ABB RAPID module: Codigo Rapid Module1

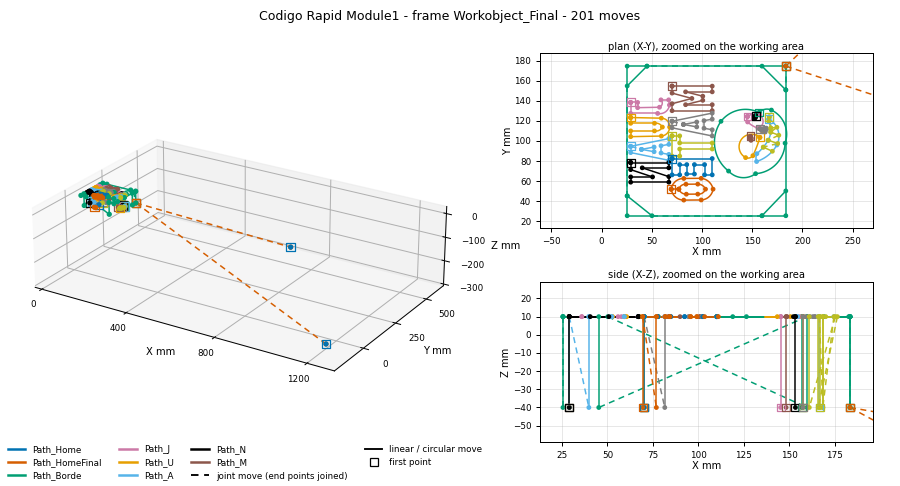
[picture p0: tool path of Codigo Rapid Module1 in frame Workobject_Final, 201 of 201 moves have a stored position in this frame; points joined in program order, loops and branches not executed]
MODULE Module1
    CONST robtarget Target_10:=[[183.5,174.5,-40],[1,0,0,0],[-2,-1,0,0],[9E+09,9E+09,9E+09,9E+09,9E+09,9E+09]];
    CONST robtarget Target_20:=[[183.5,174.5,10],[1,0,0,0],[-2,-1,0,0],[9E+09,9E+09,9E+09,9E+09,9E+09,9E+09]];
    CONST robtarget Target_30:=[[25.5,174.5,10],[1,0,0,0],[-2,-1,0,0],[9E+09,9E+09,9E+09,9E+09,9E+09,9E+09]];
    CONST robtarget Target_40:=[[25.5,25.5,10],[1,0,0,0],[-2,-1,0,0],[9E+09,9E+09,9E+09,9E+09,9E+09,9E+09]];
    CONST robtarget Target_50:=[[183.5,25.5,10],[1,0,0,0],[-2,-1,0,0],[9E+09,9E+09,9E+09,9E+09,9E+09,9E+09]];
    CONST robtarget Target_Home:=[[1257.383388943,-178.562274595,-229.244724109],[0.000082309,-0.261784185,0.00007376,-0.965126431],[0,-1,0,0],[9E+09,9E+09,9E+09,9E+09,9E+09,9E+09]];
    CONST robtarget Target_60:=[[183.5,150.793,-40],[1,0,0,0],[-2,-1,0,0],[9E+09,9E+09,9E+09,9E+09,9E+09,9E+09]];
    CONST robtarget Target_70:=[[183.5,150.793,10],[1,0,0,0],[-2,-1,0,0],[9E+09,9E+09,9E+09,9E+09,9E+09,9E+09]];
    CONST robtarget Target_80:=[[159.793,174.5,10],[1,0,0,0],[-2,-1,0,0],[9E+09,9E+09,9E+09,9E+09,9E+09,9E+09]];
    CONST robtarget Target_90:=[[45.207,174.5,-40],[1,0,0,0],[-2,-1,0,0],[9E+09,9E+09,9E+09,9E+09,9E+09,9E+09]];
    CONST robtarget Target_100:=[[45.207,174.5,10],[1,0,0,0],[-2,-1,0,0],[9E+09,9E+09,9E+09,9E+09,9E+09,9E+09]];
    CONST robtarget Target_110:=[[25.5,154.793,10],[1,0,0,0],[-2,-1,0,0],[9E+09,9E+09,9E+09,9E+09,9E+09,9E+09]];
    CONST robtarget Target_120:=[[25.5,45.24,-40],[1,0,0,0],[-2,-1,0,0],[9E+09,9E+09,9E+09,9E+09,9E+09,9E+09]];
    CONST robtarget Target_130:=[[25.5,45.24,10],[1,0,0,0],[-2,-1,0,0],[9E+09,9E+09,9E+09,9E+09,9E+09,9E+09]];
    CONST robtarget Target_140:=[[50.175,25.5,10],[1,0,0,0],[-2,-1,0,0],[9E+09,9E+09,9E+09,9E+09,9E+09,9E+09]];
    CONST robtarget Target_150:=[[159.787,25.5,-40],[1,0,0,0],[-2,-1,0,0],[9E+09,9E+09,9E+09,9E+09,9E+09,9E+09]];
    CONST robtarget Target_160:=[[159.787,25.5,10],[1,0,0,0],[-2,-1,0,0],[9E+09,9E+09,9E+09,9E+09,9E+09,9E+09]];
    CONST robtarget Target_170:=[[183.5,50.201,10],[1,0,0,0],[-2,-1,0,0],[9E+09,9E+09,9E+09,9E+09,9E+09,9E+09]];
    CONST robtarget Target_180:=[[28.978,138.344,-40],[1,0,0,0],[-2,-1,0,0],[9E+09,9E+09,9E+09,9E+09,9E+09,9E+09]];
    CONST robtarget Target_190_2:=[[28.978,138.344,10],[1,0,0,0],[0,0,0,0],[9E+09,9E+09,9E+09,9E+09,9E+09,9E+09]];
    CONST robtarget Target_200:=[[28.978,127.412,10],[1,0,0,0],[-2,-1,0,0],[9E+09,9E+09,9E+09,9E+09,9E+09,9E+09]];
    CONST robtarget Target_210:=[[55.831,127.412,10],[1,0,0,0],[-2,-1,0,0],[9E+09,9E+09,9E+09,9E+09,9E+09,9E+09]];
    CONST robtarget Target_220:=[[64.207,129.444,10],[1,0,0,0],[-2,-1,0,0],[9E+09,9E+09,9E+09,9E+09,9E+09,9E+09]];
    CONST robtarget Target_230:=[[67.563,135.757,10],[1,0,0,0],[-2,-1,0,0],[9E+09,9E+09,9E+09,9E+09,9E+09,9E+09]];
    CONST robtarget Target_240:=[[66.824,140.93,10],[1,0,0,0],[-2,-1,0,0],[9E+09,9E+09,9E+09,9E+09,9E+09,9E+09]];
    CONST robtarget Target_250:=[[59.125,140.93,10],[1,0,0,0],[-2,-1,0,0],[9E+09,9E+09,9E+09,9E+09,9E+09,9E+09]];
    CONST robtarget Target_260:=[[60.388,137.05,10],[1,0,0,0],[-2,-1,0,0],[9E+09,9E+09,9E+09,9E+09,9E+09,9E+09]];
    CONST robtarget Target_270:=[[57.678,133.57,10],[1,0,0,0],[-2,-1,0,0],[9E+09,9E+09,9E+09,9E+09,9E+09,9E+09]];
    CONST robtarget Target_280:=[[35.876,133.139,10],[1,0,0,0],[-2,-1,0,0],[9E+09,9E+09,9E+09,9E+09,9E+09,9E+09]];
    CONST robtarget Target_290:=[[35.876,138.344,10],[1,0,0,0],[-2,-1,0,0],[9E+09,9E+09,9E+09,9E+09,9E+09,9E+09]];
    CONST robtarget Target_190:=[[28.978,138.344,10],[1,0,0,0],[-2,-1,0,0],[9E+09,9E+09,9E+09,9E+09,9E+09,9E+09]];
    CONST robtarget Target_300:=[[28.978,123.316,-40],[1,0,0,0],[-2,-1,0,0],[9E+09,9E+09,9E+09,9E+09,9E+09,9E+09]];
    CONST robtarget Target_310:=[[28.978,123.316,10],[1,0,0,0],[-2,-1,0,0],[9E+09,9E+09,9E+09,9E+09,9E+09,9E+09]];
    CONST robtarget Target_320:=[[28.978,117.588,10],[1,0,0,0],[-2,-1,0,0],[9E+09,9E+09,9E+09,9E+09,9E+09,9E+09]];
    CONST robtarget Target_330:=[[52.69,117.588,10],[1,0,0,0],[-2,-1,0,0],[9E+09,9E+09,9E+09,9E+09,9E+09,9E+09]];
    CONST robtarget Target_340:=[[56.691,117.273,10],[1,0,0,0],[-2,-1,0,0],[9E+09,9E+09,9E+09,9E+09,9E+09,9E+09]];
    CONST robtarget Target_350:=[[60.542,113.801,10],[1,0,0,0],[-2,-1,0,0],[9E+09,9E+09,9E+09,9E+09,9E+09,9E+09]];
    CONST robtarget Target_360:=[[56.691,110.285,10],[1,0,0,0],[-2,-1,0,0],[9E+09,9E+09,9E+09,9E+09,9E+09,9E+09]];
    CONST robtarget Target_370:=[[52.69,109.982,10],[1,0,0,0],[-2,-1,0,0],[9E+09,9E+09,9E+09,9E+09,9E+09,9E+09]];
    CONST robtarget Target_380:=[[28.978,109.982,10],[1,0,0,0],[-2,-1,0,0],[9E+09,9E+09,9E+09,9E+09,9E+09,9E+09]];
    CONST robtarget Target_390:=[[28.978,104.254,10],[1,0,0,0],[-2,-1,0,0],[9E+09,9E+09,9E+09,9E+09,9E+09,9E+09]];
    CONST robtarget Target_400:=[[59.499,104.872,10],[1,0,0,0],[-2,-1,0,0],[9E+09,9E+09,9E+09,9E+09,9E+09,9E+09]];
    CONST robtarget Target_410:=[[65.743,108.096,10],[1,0,0,0],[-2,-1,0,0],[9E+09,9E+09,9E+09,9E+09,9E+09,9E+09]];
    CONST robtarget Target_420:=[[67.779,113.801,10],[1,0,0,0],[-2,-1,0,0],[9E+09,9E+09,9E+09,9E+09,9E+09,9E+09]];
    CONST robtarget Target_430:=[[65.743,119.791,10],[1,0,0,0],[-2,-1,0,0],[9E+09,9E+09,9E+09,9E+09,9E+09,9E+09]];
    CONST robtarget Target_440:=[[59.499,122.66,10],[1,0,0,0],[-2,-1,0,0],[9E+09,9E+09,9E+09,9E+09,9E+09,9E+09]];
    CONST robtarget Target_4101:=[[61.442,105.428,10],[1,0,0,0],[-2,-1,0,0],[9E+09,9E+09,9E+09,9E+09,9E+09,9E+09]];
    CONST robtarget Target_4301:=[[61.442,122.642,10],[1,0,0,0],[-2,-1,0,0],[9E+09,9E+09,9E+09,9E+09,9E+09,9E+09]];
    CONST robtarget Target_4000:=[[59.499,104.872,10],[1,0,0,0],[-2,-1,0,0],[9E+09,9E+09,9E+09,9E+09,9E+09,9E+09]];
    CONST robtarget Target_4400:=[[59.499,122.66,10],[1,0,0,0],[-2,-1,0,0],[9E+09,9E+09,9E+09,9E+09,9E+09,9E+09]];
    CONST robtarget Target_4300:=[[65.743,119.791,10],[1,0,0,0],[-2,-1,0,0],[9E+09,9E+09,9E+09,9E+09,9E+09,9E+09]];
    CONST robtarget Target_4100:=[[65.743,108.096,10],[1,0,0,0],[-2,-1,0,0],[9E+09,9E+09,9E+09,9E+09,9E+09,9E+09]];
    CONST robtarget Target_450:=[[28.978,94.616,-40],[1,0,0,0],[-2,-1,0,0],[9E+09,9E+09,9E+09,9E+09,9E+09,9E+09]];
    CONST robtarget Target_460:=[[28.978,94.616,10],[1,0,0,0],[-2,-1,0,0],[9E+09,9E+09,9E+09,9E+09,9E+09,9E+09]];
    CONST robtarget Target_470:=[[28.978,88.395,10],[1,0,0,0],[-2,-1,0,0],[9E+09,9E+09,9E+09,9E+09,9E+09,9E+09]];
    CONST robtarget Target_480:=[[66.978,80.697,10],[1,0,0,0],[-2,-1,0,0],[9E+09,9E+09,9E+09,9E+09,9E+09,9E+09]];
    CONST robtarget Target_490:=[[66.978,86.579,10],[1,0,0,0],[-2,-1,0,0],[9E+09,9E+09,9E+09,9E+09,9E+09,9E+09]];
    CONST robtarget Target_500:=[[59.218,87.995,10],[1,0,0,0],[-2,-1,0,0],[9E+09,9E+09,9E+09,9E+09,9E+09,9E+09]];
    CONST robtarget Target_510:=[[59.218,95.17,10],[1,0,0,0],[-2,-1,0,0],[9E+09,9E+09,9E+09,9E+09,9E+09,9E+09]];
    CONST robtarget Target_520:=[[66.978,96.587,10],[1,0,0,0],[-2,-1,0,0],[9E+09,9E+09,9E+09,9E+09,9E+09,9E+09]];
    CONST robtarget Target_530:=[[66.978,102.314,10],[1,0,0,0],[-2,-1,0,0],[9E+09,9E+09,9E+09,9E+09,9E+09,9E+09]];
    CONST robtarget Target_540:=[[39.756,91.598,-40],[1,0,0,0],[-2,-1,0,0],[9E+09,9E+09,9E+09,9E+09,9E+09,9E+09]];
    CONST robtarget Target_550:=[[39.756,91.598,10],[1,0,0,0],[-2,-1,0,0],[9E+09,9E+09,9E+09,9E+09,9E+09,9E+09]];
    CONST robtarget Target_560:=[[52.32,89.258,10],[1,0,0,0],[-2,-1,0,0],[9E+09,9E+09,9E+09,9E+09,9E+09,9E+09]];
    CONST robtarget Target_570:=[[52.32,93.908,10],[1,0,0,0],[-2,-1,0,0],[9E+09,9E+09,9E+09,9E+09,9E+09,9E+09]];
    CONST robtarget Target_580:=[[28.978,78.449,-40],[1,0,0,0],[-2,-1,0,0],[9E+09,9E+09,9E+09,9E+09,9E+09,9E+09]];
    CONST robtarget Target_590:=[[28.978,78.449,10],[1,0,0,0],[-2,-1,0,0],[9E+09,9E+09,9E+09,9E+09,9E+09,9E+09]];
    CONST robtarget Target_600:=[[28.978,71.428,10],[1,0,0,0],[-2,-1,0,0],[9E+09,9E+09,9E+09,9E+09,9E+09,9E+09]];
    CONST robtarget Target_610:=[[50.749,64.16,10],[1,0,0,0],[-2,-1,0,0],[9E+09,9E+09,9E+09,9E+09,9E+09,9E+09]];
    CONST robtarget Target_620:=[[28.978,64.16,10],[1,0,0,0],[-2,-1,0,0],[9E+09,9E+09,9E+09,9E+09,9E+09,9E+09]];
    CONST robtarget Target_630:=[[28.978,58.925,10],[1,0,0,0],[-2,-1,0,0],[9E+09,9E+09,9E+09,9E+09,9E+09,9E+09]];
    CONST robtarget Target_640:=[[66.978,58.925,10],[1,0,0,0],[-2,-1,0,0],[9E+09,9E+09,9E+09,9E+09,9E+09,9E+09]];
    CONST robtarget Target_650:=[[66.978,64.438,10],[1,0,0,0],[-2,-1,0,0],[9E+09,9E+09,9E+09,9E+09,9E+09,9E+09]];
    CONST robtarget Target_660:=[[40.495,73.214,10],[1,0,0,0],[-2,-1,0,0],[9E+09,9E+09,9E+09,9E+09,9E+09,9E+09]];
    CONST robtarget Target_670:=[[66.978,73.214,10],[1,0,0,0],[-2,-1,0,0],[9E+09,9E+09,9E+09,9E+09,9E+09,9E+09]];
    CONST robtarget Target_680:=[[66.978,78.449,10],[1,0,0,0],[-2,-1,0,0],[9E+09,9E+09,9E+09,9E+09,9E+09,9E+09]];
    CONST robtarget Target_690:=[[70.192,154.588,-40],[1,0,0,0],[-2,-1,0,0],[9E+09,9E+09,9E+09,9E+09,9E+09,9E+09]];
    CONST robtarget Target_700:=[[70.192,154.588,10],[1,0,0,0],[-2,-1,0,0],[9E+09,9E+09,9E+09,9E+09,9E+09,9E+09]];
    CONST robtarget Target_710:=[[70.192,147.651,10],[1,0,0,0],[-2,-1,0,0],[9E+09,9E+09,9E+09,9E+09,9E+09,9E+09]];
    CONST robtarget Target_720:=[[89.932,142.335,10],[1,0,0,0],[-2,-1,0,0],[9E+09,9E+09,9E+09,9E+09,9E+09,9E+09]];
    CONST robtarget Target_730:=[[70.192,137.051,10],[1,0,0,0],[-2,-1,0,0],[9E+09,9E+09,9E+09,9E+09,9E+09,9E+09]];
    CONST robtarget Target_740:=[[70.192,130.115,10],[1,0,0,0],[-2,-1,0,0],[9E+09,9E+09,9E+09,9E+09,9E+09,9E+09]];
    CONST robtarget Target_750:=[[110.192,130.115,10],[1,0,0,0],[-2,-1,0,0],[9E+09,9E+09,9E+09,9E+09,9E+09,9E+09]];
    CONST robtarget Target_760:=[[110.192,136.111,10],[1,0,0,0],[-2,-1,0,0],[9E+09,9E+09,9E+09,9E+09,9E+09,9E+09]];
    CONST robtarget Target_770:=[[83.676,136.111,10],[1,0,0,0],[-2,-1,0,0],[9E+09,9E+09,9E+09,9E+09,9E+09,9E+09]];
    CONST robtarget Target_780:=[[100.791,140.455,10],[1,0,0,0],[-2,-1,0,0],[9E+09,9E+09,9E+09,9E+09,9E+09,9E+09]];
    CONST robtarget Target_790:=[[100.791,144.572,10],[1,0,0,0],[-2,-1,0,0],[9E+09,9E+09,9E+09,9E+09,9E+09,9E+09]];
    CONST robtarget Target_800:=[[83.676,148.915,10],[1,0,0,0],[-2,-1,0,0],[9E+09,9E+09,9E+09,9E+09,9E+09,9E+09]];
    CONST robtarget Target_810:=[[110.192,148.915,10],[1,0,0,0],[-2,-1,0,0],[9E+09,9E+09,9E+09,9E+09,9E+09,9E+09]];
    CONST robtarget Target_820:=[[110.192,154.588,10],[1,0,0,0],[-2,-1,0,0],[9E+09,9E+09,9E+09,9E+09,9E+09,9E+09]];
    CONST robtarget Target_830:=[[70.192,119.612,-40],[1,0,0,0],[-2,-1,0,0],[9E+09,9E+09,9E+09,9E+09,9E+09,9E+09]];
    CONST robtarget Target_840:=[[70.192,119.612,10],[1,0,0,0],[-2,-1,0,0],[9E+09,9E+09,9E+09,9E+09,9E+09,9E+09]];
    CONST robtarget Target_850:=[[70.192,113.064,10],[1,0,0,0],[-2,-1,0,0],[9E+09,9E+09,9E+09,9E+09,9E+09,9E+09]];
    CONST robtarget Target_860:=[[110.192,104.961,10],[1,0,0,0],[-2,-1,0,0],[9E+09,9E+09,9E+09,9E+09,9E+09,9E+09]];
    CONST robtarget Target_870:=[[110.192,111.152,10],[1,0,0,0],[-2,-1,0,0],[9E+09,9E+09,9E+09,9E+09,9E+09,9E+09]];
    CONST robtarget Target_880:=[[102.023,112.643,10],[1,0,0,0],[-2,-1,0,0],[9E+09,9E+09,9E+09,9E+09,9E+09,9E+09]];
    CONST robtarget Target_890:=[[102.023,120.196,10],[1,0,0,0],[-2,-1,0,0],[9E+09,9E+09,9E+09,9E+09,9E+09,9E+09]];
    CONST robtarget Target_900:=[[110.192,121.687,10],[1,0,0,0],[-2,-1,0,0],[9E+09,9E+09,9E+09,9E+09,9E+09,9E+09]];
    CONST robtarget Target_910:=[[110.192,127.716,10],[1,0,0,0],[-2,-1,0,0],[9E+09,9E+09,9E+09,9E+09,9E+09,9E+09]];
    CONST robtarget Target_920:=[[81.537,116.436,-40],[1,0,0,0],[-2,-1,0,0],[9E+09,9E+09,9E+09,9E+09,9E+09,9E+09]];
    CONST robtarget Target_930:=[[81.537,116.436,10],[1,0,0,0],[-2,-1,0,0],[9E+09,9E+09,9E+09,9E+09,9E+09,9E+09]];
    CONST robtarget Target_940:=[[94.762,113.972,10],[1,0,0,0],[-2,-1,0,0],[9E+09,9E+09,9E+09,9E+09,9E+09,9E+09]];
    CONST robtarget Target_950:=[[94.762,118.867,10],[1,0,0,0],[-2,-1,0,0],[9E+09,9E+09,9E+09,9E+09,9E+09,9E+09]];
    CONST robtarget Target_960:=[[70.192,105.058,-40],[1,0,0,0],[-2,-1,0,0],[9E+09,9E+09,9E+09,9E+09,9E+09,9E+09]];
    CONST robtarget Target_970:=[[70.192,105.058,10],[1,0,0,0],[-2,-1,0,0],[9E+09,9E+09,9E+09,9E+09,9E+09,9E+09]];
    CONST robtarget Target_980:=[[70.192,84.896,10],[1,0,0,0],[-2,-1,0,0],[9E+09,9E+09,9E+09,9E+09,9E+09,9E+09]];
    CONST robtarget Target_990:=[[77.809,84.896,10],[1,0,0,0],[-2,-1,0,0],[9E+09,9E+09,9E+09,9E+09,9E+09,9E+09]];
    CONST robtarget Target_1000:=[[77.809,91.962,10],[1,0,0,0],[-2,-1,0,0],[9E+09,9E+09,9E+09,9E+09,9E+09,9E+09]];
    CONST robtarget Target_1010:=[[110.192,91.962,10],[1,0,0,0],[-2,-1,0,0],[9E+09,9E+09,9E+09,9E+09,9E+09,9E+09]];
    CONST robtarget Target_1020:=[[110.192,97.991,10],[1,0,0,0],[-2,-1,0,0],[9E+09,9E+09,9E+09,9E+09,9E+09,9E+09]];
    CONST robtarget Target_1030:=[[77.809,97.991,10],[1,0,0,0],[-2,-1,0,0],[9E+09,9E+09,9E+09,9E+09,9E+09,9E+09]];
    CONST robtarget Target_1040:=[[77.809,105.058,10],[1,0,0,0],[-2,-1,0,0],[9E+09,9E+09,9E+09,9E+09,9E+09,9E+09]];
    CONST robtarget Target_1050:=[[70.192,82.432,-40],[1,0,0,0],[-2,-1,0,0],[9E+09,9E+09,9E+09,9E+09,9E+09,9E+09]];
    CONST robtarget Target_1060:=[[70.192,82.432,10],[1,0,0,0],[-2,-1,0,0],[9E+09,9E+09,9E+09,9E+09,9E+09,9E+09]];
    CONST robtarget Target_1070:=[[70.192,66.225,10],[1,0,0,0],[-2,-1,0,0],[9E+09,9E+09,9E+09,9E+09,9E+09,9E+09]];
    CONST robtarget Target_1080:=[[77.809,66.225,10],[1,0,0,0],[-2,-1,0,0],[9E+09,9E+09,9E+09,9E+09,9E+09,9E+09]];
    CONST robtarget Target_1090:=[[77.809,76.436,10],[1,0,0,0],[-2,-1,0,0],[9E+09,9E+09,9E+09,9E+09,9E+09,9E+09]];
    CONST robtarget Target_1100:=[[84.843,76.436,10],[1,0,0,0],[-2,-1,0,0],[9E+09,9E+09,9E+09,9E+09,9E+09,9E+09]];
    CONST robtarget Target_1110:=[[84.843,67.035,10],[1,0,0,0],[-2,-1,0,0],[9E+09,9E+09,9E+09,9E+09,9E+09,9E+09]];
    CONST robtarget Target_1120:=[[92.461,67.035,10],[1,0,0,0],[-2,-1,0,0],[9E+09,9E+09,9E+09,9E+09,9E+09,9E+09]];
    CONST robtarget Target_1130:=[[92.461,76.436,10],[1,0,0,0],[-2,-1,0,0],[9E+09,9E+09,9E+09,9E+09,9E+09,9E+09]];
    CONST robtarget Target_1140:=[[102.574,76.436,10],[1,0,0,0],[-2,-1,0,0],[9E+09,9E+09,9E+09,9E+09,9E+09,9E+09]];
    CONST robtarget Target_1150:=[[102.574,66.225,10],[1,0,0,0],[-2,-1,0,0],[9E+09,9E+09,9E+09,9E+09,9E+09,9E+09]];
    CONST robtarget Target_1160:=[[110.192,66.225,10],[1,0,0,0],[-2,-1,0,0],[9E+09,9E+09,9E+09,9E+09,9E+09,9E+09]];
    CONST robtarget Target_1170:=[[110.192,82.432,10],[1,0,0,0],[-2,-1,0,0],[9E+09,9E+09,9E+09,9E+09,9E+09,9E+09]];
    CONST robtarget Target_1180:=[[69.349,51.962,-40],[1,0,0,0],[-2,-1,0,0],[9E+09,9E+09,9E+09,9E+09,9E+09,9E+09]];
    CONST robtarget Target_1190:=[[69.349,51.962,10],[1,0,0,0],[-2,-1,0,0],[9E+09,9E+09,9E+09,9E+09,9E+09,9E+09]];
    CONST robtarget Target_1200:=[[72.94,44.787,10],[1,0,0,0],[-2,-1,0,0],[9E+09,9E+09,9E+09,9E+09,9E+09,9E+09]];
    CONST robtarget Target_1210:=[[81.874,41.067,10],[1,0,0,0],[-2,-1,0,0],[9E+09,9E+09,9E+09,9E+09,9E+09,9E+09]];
    CONST robtarget Target_1220:=[[99.202,41.204,10],[1,0,0,0],[-2,-1,0,0],[9E+09,9E+09,9E+09,9E+09,9E+09,9E+09]];
    CONST robtarget Target_1230:=[[107.314,44.677,10],[1,0,0,0],[-2,-1,0,0],[9E+09,9E+09,9E+09,9E+09,9E+09,9E+09]];
    CONST robtarget Target_1240:=[[111.034,51.962,10],[1,0,0,0],[-2,-1,0,0],[9E+09,9E+09,9E+09,9E+09,9E+09,9E+09]];
    CONST robtarget Target_1250:=[[107.314,58.928,10],[1,0,0,0],[-2,-1,0,0],[9E+09,9E+09,9E+09,9E+09,9E+09,9E+09]];
    CONST robtarget Target_1260:=[[99.202,62.766,10],[1,0,0,0],[-2,-1,0,0],[9E+09,9E+09,9E+09,9E+09,9E+09,9E+09]];
    CONST robtarget Target_1270:=[[81.874,62.635,10],[1,0,0,0],[-2,-1,0,0],[9E+09,9E+09,9E+09,9E+09,9E+09,9E+09]];
    CONST robtarget Target_1280:=[[72.94,59.1,10],[1,0,0,0],[-2,-1,0,0],[9E+09,9E+09,9E+09,9E+09,9E+09,9E+09]];
    CONST robtarget Target_1290:=[[76.902,51.962,-40],[1,0,0,0],[-2,-1,0,0],[9E+09,9E+09,9E+09,9E+09,9E+09,9E+09]];
    CONST robtarget Target_1300:=[[76.902,51.962,10],[1,0,0,0],[-2,-1,0,0],[9E+09,9E+09,9E+09,9E+09,9E+09,9E+09]];
    CONST robtarget Target_1310:=[[79.981,48.202,10],[1,0,0,0],[-2,-1,0,0],[9E+09,9E+09,9E+09,9E+09,9E+09,9E+09]];
    CONST robtarget Target_1320:=[[84.396,46.967,10],[1,0,0,0],[-2,-1,0,0],[9E+09,9E+09,9E+09,9E+09,9E+09,9E+09]];
    CONST robtarget Target_1330:=[[95.811,47.035,10],[1,0,0,0],[-2,-1,0,0],[9E+09,9E+09,9E+09,9E+09,9E+09,9E+09]];
    CONST robtarget Target_1340:=[[100.073,47.88,10],[1,0,0,0],[-2,-1,0,0],[9E+09,9E+09,9E+09,9E+09,9E+09,9E+09]];
    CONST robtarget Target_1350:=[[103.482,51.962,10],[1,0,0,0],[-2,-1,0,0],[9E+09,9E+09,9E+09,9E+09,9E+09,9E+09]];
    CONST robtarget Target_1360:=[[100.073,55.865,10],[1,0,0,0],[-2,-1,0,0],[9E+09,9E+09,9E+09,9E+09,9E+09,9E+09]];
    CONST robtarget Target_1370:=[[95.811,56.99,10],[1,0,0,0],[-2,-1,0,0],[9E+09,9E+09,9E+09,9E+09,9E+09,9E+09]];
    CONST robtarget Target_1380:=[[84.063,56.892,10],[1,0,0,0],[-2,-1,0,0],[9E+09,9E+09,9E+09,9E+09,9E+09,9E+09]];
    CONST robtarget Target_1390:=[[78.981,55.17,10],[1,0,0,0],[-2,-1,0,0],[9E+09,9E+09,9E+09,9E+09,9E+09,9E+09]];
    CONST robtarget Target_1400:=[[156.983,128.308,-40],[1,0,0,0],[-2,-1,0,0],[9E+09,9E+09,9E+09,9E+09,9E+09,9E+09]];
    CONST robtarget Target_1410:=[[156.983,128.308,10],[1,0,0,0],[-2,-1,0,0],[9E+09,9E+09,9E+09,9E+09,9E+09,9E+09]];
    CONST robtarget Target_1420:=[[136.354,130.668,10],[1,0,0,0],[-2,-1,0,0],[9E+09,9E+09,9E+09,9E+09,9E+09,9E+09]];
    CONST robtarget Target_1430:=[[118.934,119.56,10],[1,0,0,0],[-2,-1,0,0],[9E+09,9E+09,9E+09,9E+09,9E+09,9E+09]];
    CONST robtarget Target_1440:=[[113.201,91.153,10],[1,0,0,0],[-2,-1,0,0],[9E+09,9E+09,9E+09,9E+09,9E+09,9E+09]];
    CONST robtarget Target_1450:=[[126.483,69.994,10],[1,0,0,0],[-2,-1,0,0],[9E+09,9E+09,9E+09,9E+09,9E+09,9E+09]];
    CONST robtarget Target_1460:=[[139.823,63.474,10],[1,0,0,0],[-2,-1,0,0],[9E+09,9E+09,9E+09,9E+09,9E+09,9E+09]];
    CONST robtarget Target_1470:=[[153.393,67.379,10],[1,0,0,0],[-2,-1,0,0],[9E+09,9E+09,9E+09,9E+09,9E+09,9E+09]];
    CONST robtarget Target_1480:=[[167.51,71.819,10],[1,0,0,0],[-2,-1,0,0],[9E+09,9E+09,9E+09,9E+09,9E+09,9E+09]];
    CONST robtarget Target_1490:=[[182.795,97.789,10],[1,0,0,0],[-2,-1,0,0],[9E+09,9E+09,9E+09,9E+09,9E+09,9E+09]];
    CONST robtarget Target_1500:=[[179.202,122.449,10],[1,0,0,0],[-2,-1,0,0],[9E+09,9E+09,9E+09,9E+09,9E+09,9E+09]];
    CONST robtarget Target_1510:=[[169.163,130.753,10],[1,0,0,0],[-2,-1,0,0],[9E+09,9E+09,9E+09,9E+09,9E+09,9E+09]];
    CONST robtarget Target_1540:=[[145.319,124.3,10],[1,0,0,0],[-2,-1,0,0],[9E+09,9E+09,9E+09,9E+09,9E+09,9E+09]];
    CONST robtarget Target_1520:=[[164.258,131.707,10],[1,0,0,0],[-2,-1,0,0],[9E+09,9E+09,9E+09,9E+09,9E+09,9E+09]];
    CONST robtarget Target_1530:=[[145.319,124.3,-40],[1,0,0,0],[-2,-1,0,0],[9E+09,9E+09,9E+09,9E+09,9E+09,9E+09]];
    CONST robtarget Target_1550:=[[144.635,121.725,10],[1,0,0,0],[-2,-1,0,0],[9E+09,9E+09,9E+09,9E+09,9E+09,9E+09]];
    CONST robtarget Target_1560:=[[145.446,118.91,10],[1,0,0,0],[-2,-1,0,0],[9E+09,9E+09,9E+09,9E+09,9E+09,9E+09]];
    CONST robtarget Target_1570:=[[151.071,114.797,10],[1,0,0,0],[-2,-1,0,0],[9E+09,9E+09,9E+09,9E+09,9E+09,9E+09]];
    CONST robtarget Target_1580:=[[155.76,112.62,10],[1,0,0,0],[-2,-1,0,0],[9E+09,9E+09,9E+09,9E+09,9E+09,9E+09]];
    CONST robtarget Target_1590:=[[160.801,118.423,10],[1,0,0,0],[-2,-1,0,0],[9E+09,9E+09,9E+09,9E+09,9E+09,9E+09]];
    CONST robtarget Target_1600:=[[157.663,125.533,10],[1,0,0,0],[-2,-1,0,0],[9E+09,9E+09,9E+09,9E+09,9E+09,9E+09]];
    CONST robtarget Target_1610:=[[151.045,126.726,10],[1,0,0,0],[-2,-1,0,0],[9E+09,9E+09,9E+09,9E+09,9E+09,9E+09]];
    CONST robtarget Target_1620:=[[157.652,103.483,-40],[1,0,0,0],[-2,-1,0,0],[9E+09,9E+09,9E+09,9E+09,9E+09,9E+09]];
    CONST robtarget Target_1630:=[[157.652,103.483,10],[1,0,0,0],[-2,-1,0,0],[9E+09,9E+09,9E+09,9E+09,9E+09,9E+09]];
    CONST robtarget Target_1640:=[[138.076,99.514,10],[1,0,0,0],[-2,-1,0,0],[9E+09,9E+09,9E+09,9E+09,9E+09,9E+09]];
    CONST robtarget Target_1650:=[[143.464,83.388,10],[1,0,0,0],[-2,-1,0,0],[9E+09,9E+09,9E+09,9E+09,9E+09,9E+09]];
    CONST robtarget Target_1660:=[[147.351,83.085,10],[1,0,0,0],[-2,-1,0,0],[9E+09,9E+09,9E+09,9E+09,9E+09,9E+09]];
    CONST robtarget Target_1670:=[[150.699,85.338,10],[1,0,0,0],[-2,-1,0,0],[9E+09,9E+09,9E+09,9E+09,9E+09,9E+09]];
    CONST robtarget Target_1680:=[[154.139,93.197,10],[1,0,0,0],[-2,-1,0,0],[9E+09,9E+09,9E+09,9E+09,9E+09,9E+09]];
    CONST robtarget Target_1690:=[[166.684,121.689,-40],[1,0,0,0],[-2,-1,0,0],[9E+09,9E+09,9E+09,9E+09,9E+09,9E+09]];
    CONST robtarget Target_1700:=[[166.684,121.689,10],[1,0,0,0],[-2,-1,0,0],[9E+09,9E+09,9E+09,9E+09,9E+09,9E+09]];
    CONST robtarget Target_1710:=[[168.683,110.823,10],[1,0,0,0],[-2,-1,0,0],[9E+09,9E+09,9E+09,9E+09,9E+09,9E+09]];
    CONST robtarget Target_1720:=[[165.783,100.387,10],[1,0,0,0],[-2,-1,0,0],[9E+09,9E+09,9E+09,9E+09,9E+09,9E+09]];
    CONST robtarget Target_1730:=[[160.867,93.548,10],[1,0,0,0],[-2,-1,0,0],[9E+09,9E+09,9E+09,9E+09,9E+09,9E+09]];
    CONST robtarget Target_1740:=[[154.691,87.305,10],[1,0,0,0],[-2,-1,0,0],[9E+09,9E+09,9E+09,9E+09,9E+09,9E+09]];
    CONST robtarget Target_1750:=[[153.8,83.479,10],[1,0,0,0],[-2,-1,0,0],[9E+09,9E+09,9E+09,9E+09,9E+09,9E+09]];
    CONST robtarget Target_1760:=[[154.401,79.5,10],[1,0,0,0],[-2,-1,0,0],[9E+09,9E+09,9E+09,9E+09,9E+09,9E+09]];
    CONST robtarget Target_1770:=[[167.265,86.892,10],[1,0,0,0],[-2,-1,0,0],[9E+09,9E+09,9E+09,9E+09,9E+09,9E+09]];
    CONST robtarget Target_1780:=[[174.643,95.985,10],[1,0,0,0],[-2,-1,0,0],[9E+09,9E+09,9E+09,9E+09,9E+09,9E+09]];
    CONST robtarget Target_1790:=[[175.81,110.356,10],[1,0,0,0],[-2,-1,0,0],[9E+09,9E+09,9E+09,9E+09,9E+09,9E+09]];
    CONST robtarget Target_1800:=[[153.457,125.06,-40],[1,0,0,0],[-2,-1,0,0],[9E+09,9E+09,9E+09,9E+09,9E+09,9E+09]];
    CONST robtarget Target_1810:=[[153.457,125.06,10],[1,0,0,0],[-2,-1,0,0],[9E+09,9E+09,9E+09,9E+09,9E+09,9E+09]];
    CONST robtarget Target_1820:=[[150.736,124.071,10],[1,0,0,0],[-2,-1,0,0],[9E+09,9E+09,9E+09,9E+09,9E+09,9E+09]];
    CONST robtarget Target_1830:=[[152.376,122.188,10],[1,0,0,0],[-2,-1,0,0],[9E+09,9E+09,9E+09,9E+09,9E+09,9E+09]];
    CONST robtarget Target_1840:=[[155.037,123.546,10],[1,0,0,0],[-2,-1,0,0],[9E+09,9E+09,9E+09,9E+09,9E+09,9E+09]];
    CONST robtarget Target_1850:=[[148.32,104.491,-40],[1,0,0,0],[-2,-1,0,0],[9E+09,9E+09,9E+09,9E+09,9E+09,9E+09]];
    CONST robtarget Target_1860:=[[148.32,104.491,10],[1,0,0,0],[-2,-1,0,0],[9E+09,9E+09,9E+09,9E+09,9E+09,9E+09]];
    CONST robtarget Target_1870:=[[146.377,102.441,10],[1,0,0,0],[-2,-1,0,0],[9E+09,9E+09,9E+09,9E+09,9E+09,9E+09]];
    CONST robtarget Target_1880:=[[148.838,100.636,10],[1,0,0,0],[-2,-1,0,0],[9E+09,9E+09,9E+09,9E+09,9E+09,9E+09]];
    CONST robtarget Target_1890:=[[150.781,103.034,10],[1,0,0,0],[-2,-1,0,0],[9E+09,9E+09,9E+09,9E+09,9E+09,9E+09]];
    CONST robtarget Target_1900:=[[157.666,111.998,-40],[1,0,0,0],[-2,-1,0,0],[9E+09,9E+09,9E+09,9E+09,9E+09,9E+09]];
    CONST robtarget Target_1910:=[[157.666,111.998,10],[1,0,0,0],[-2,-1,0,0],[9E+09,9E+09,9E+09,9E+09,9E+09,9E+09]];
    CONST robtarget Target_1920:=[[158.56,110.911,10],[1,0,0,0],[-2,-1,0,0],[9E+09,9E+09,9E+09,9E+09,9E+09,9E+09]];
    CONST robtarget Target_1930:=[[159.572,110.107,10],[1,0,0,0],[-2,-1,0,0],[9E+09,9E+09,9E+09,9E+09,9E+09,9E+09]];
    CONST robtarget Target_1940:=[[161.52,109.307,10],[1,0,0,0],[-2,-1,0,0],[9E+09,9E+09,9E+09,9E+09,9E+09,9E+09]];
    CONST robtarget Target_1950:=[[163.009,108.881,10],[1,0,0,0],[-2,-1,0,0],[9E+09,9E+09,9E+09,9E+09,9E+09,9E+09]];
    CONST robtarget Target_1960:=[[163.866,110.235,10],[1,0,0,0],[-2,-1,0,0],[9E+09,9E+09,9E+09,9E+09,9E+09,9E+09]];
    CONST robtarget Target_1970:=[[164.178,111.356,10],[1,0,0,0],[-2,-1,0,0],[9E+09,9E+09,9E+09,9E+09,9E+09,9E+09]];
    CONST robtarget Target_1980:=[[164.587,112.208,10],[1,0,0,0],[-2,-1,0,0],[9E+09,9E+09,9E+09,9E+09,9E+09,9E+09]];
    CONST robtarget Target_1990:=[[164.093,112.759,10],[1,0,0,0],[-2,-1,0,0],[9E+09,9E+09,9E+09,9E+09,9E+09,9E+09]];
    CONST robtarget Target_2000:=[[163.273,112.996,10],[1,0,0,0],[-2,-1,0,0],[9E+09,9E+09,9E+09,9E+09,9E+09,9E+09]];
    CONST robtarget Target_2010:=[[161.42,112.403,10],[1,0,0,0],[-2,-1,0,0],[9E+09,9E+09,9E+09,9E+09,9E+09,9E+09]];
    CONST robtarget Target_2020:=[[159.441,111.994,10],[1,0,0,0],[-2,-1,0,0],[9E+09,9E+09,9E+09,9E+09,9E+09,9E+09]];
    CONST robtarget Target_2030:=[[167.07,123.958,-40],[1,0,0,0],[-2,-1,0,0],[9E+09,9E+09,9E+09,9E+09,9E+09,9E+09]];
    CONST robtarget Target_2040:=[[167.07,123.958,10],[1,0,0,0],[-2,-1,0,0],[9E+09,9E+09,9E+09,9E+09,9E+09,9E+09]];
    CONST robtarget Target_2050:=[[166.593,119.422,10],[1,0,0,0],[-2,-1,0,0],[9E+09,9E+09,9E+09,9E+09,9E+09,9E+09]];
    CONST robtarget Target_2060:=[[168.567,112.837,-40],[1,0,0,0],[-2,-1,0,0],[9E+09,9E+09,9E+09,9E+09,9E+09,9E+09]];
    CONST robtarget Target_2070:=[[168.567,112.837,10],[1,0,0,0],[-2,-1,0,0],[9E+09,9E+09,9E+09,9E+09,9E+09,9E+09]];
    CONST robtarget Target_2070B:=[[174.612,113.629,10],[1,0,0,0],[-2,-1,0,0],[9E+09,9E+09,9E+09,9E+09,9E+09,9E+09]];
    CONST robtarget Target_2080:=[[168.496,108.759,-40],[1,0,0,0],[-2,-1,0,0],[9E+09,9E+09,9E+09,9E+09,9E+09,9E+09]];
    CONST robtarget Target_2090:=[[168.496,108.759,10],[1,0,0,0],[-2,-1,0,0],[9E+09,9E+09,9E+09,9E+09,9E+09,9E+09]];
    CONST robtarget Target_2100:=[[176.542,105.68,10],[1,0,0,0],[-2,-1,0,0],[9E+09,9E+09,9E+09,9E+09,9E+09,9E+09]];
    CONST robtarget Target_2110:=[[165.999,100.739,-40],[1,0,0,0],[-2,-1,0,0],[9E+09,9E+09,9E+09,9E+09,9E+09,9E+09]];
    CONST robtarget Target_2120:=[[165.999,100.739,10],[1,0,0,0],[-2,-1,0,0],[9E+09,9E+09,9E+09,9E+09,9E+09,9E+09]];
    CONST robtarget Target_2130:=[[175.437,97.449,10],[1,0,0,0],[-2,-1,0,0],[9E+09,9E+09,9E+09,9E+09,9E+09,9E+09]];
    CONST robtarget Target_2140:=[[161.076,93.799,-40],[1,0,0,0],[-2,-1,0,0],[9E+09,9E+09,9E+09,9E+09,9E+09,9E+09]];
    CONST robtarget Target_2150:=[[161.076,93.799,10],[1,0,0,0],[-2,-1,0,0],[9E+09,9E+09,9E+09,9E+09,9E+09,9E+09]];
    CONST robtarget Target_2160:=[[170.117,89.729,10],[1,0,0,0],[-2,-1,0,0],[9E+09,9E+09,9E+09,9E+09,9E+09,9E+09]];
    CONST robtarget Target_Mantenimiento:=[[639.866190191,608.287132031,-287.300908579],[0.627348755,-0.364990812,-0.326503552,-0.605483837],[-2,0,-1,0],[9E+09,9E+09,9E+09,9E+09,9E+09,9E+09]];
    !***********************************************************



    PROC main()

        WHILE TRUE DO
        IF DI_01=1 THEN
            Path_Home;
            Set DO_01;
            Set FWD_Conveyor;
            Set BWD_Conveyor;
            WaitTime 3;
            Reset BWD_Conveyor;
            Reset FWD_Conveyor;
            Reset DO_01;
        ENDIF
        IF DI_02=1 THEN
            Set DO_02;
            Path_Mantenimiento;
            Reset DO_02;
        ENDIF
        IF DI_03=1 THEN
            Set DO_03;
            Set FWD_Conveyor;
            WaitTime 3;
            Reset FWD_Conveyor;
            !Path_Borde;#Se Hizo el Borde del dibujo para la caja pero por cuestiones de seguridad de la herramienta en fisico se Obta por no ejecutar esta linea
            Path_J;
            Path_U;
            Path_A;
            Path_N;
            Path_M;
            Path_A2;
            Path_T;
            Path_E;
            Path_0;
            Path_SansBorde;
            Path_Sans_OJO1;
            Path_Sans_OJO2;
            Path_SansBoca;
            Path_SansPUPILA1;
            Path_SansPUPILA2;
            Path_SansNariz;
            Path_SansDientes;
            Path_Mantenimiento2;
            Set FWD_Conveyor;
            WaitTime 3;
            Reset FWD_Conveyor;
            Reset DO_03;
            Path_Home;
        ENDIF
        ENDWHILE



    ENDPROC
    PROC Path_Home()
        MoveJ Target_Home,v200,z1,HerramientaFinal\WObj:=Workobject_Final;

    ENDPROC
    PROC Path_HomeFinal()
        MoveL Target_10,v200,z1,HerramientaFinal\WObj:=Workobject_Final;
        MoveJ Target_Home,v200,z1,HerramientaFinal\WObj:=Workobject_Final;

    ENDPROC
    PROC Path_Borde()
        MoveJ Target_10,v200,z1,HerramientaFinal\WObj:=Workobject_Final;
        MoveL Target_20,v100,z1,HerramientaFinal\WObj:=Workobject_Final;
        MoveL Target_30,v100,z1,HerramientaFinal\WObj:=Workobject_Final;
        MoveL Target_40,v100,z1,HerramientaFinal\WObj:=Workobject_Final;
        MoveL Target_50,v100,z1,HerramientaFinal\WObj:=Workobject_Final;
        MoveL Target_20,v100,z1,HerramientaFinal\WObj:=Workobject_Final;
        MoveJ Target_60,v100,z1,HerramientaFinal\WObj:=Workobject_Final;
        MoveL Target_70,v100,z1,HerramientaFinal\WObj:=Workobject_Final;
        MoveL Target_80,v100,z1,HerramientaFinal\WObj:=Workobject_Final;
        MoveJ Target_90,v100,z1,HerramientaFinal\WObj:=Workobject_Final;
        MoveL Target_100,v100,z1,HerramientaFinal\WObj:=Workobject_Final;
        MoveL Target_110,v100,z1,HerramientaFinal\WObj:=Workobject_Final;
        MoveJ Target_120,v100,z1,HerramientaFinal\WObj:=Workobject_Final;
        MoveL Target_130,v100,z1,HerramientaFinal\WObj:=Workobject_Final;
        MoveL Target_140,v100,z1,HerramientaFinal\WObj:=Workobject_Final;
        MoveJ Target_150,v100,z1,HerramientaFinal\WObj:=Workobject_Final;
        MoveL Target_160,v100,z1,HerramientaFinal\WObj:=Workobject_Final;
        MoveL Target_170,v100,z1,HerramientaFinal\WObj:=Workobject_Final;
    ENDPROC
    PROC Path_J()
        MoveJ Target_180,v200,z1,HerramientaFinal\WObj:=Workobject_Final;
        MoveL Target_190,v100,z1,HerramientaFinal\WObj:=Workobject_Final;
        MoveL Target_200,v100,z1,HerramientaFinal\WObj:=Workobject_Final;
        MoveL Target_210,v100,z1,HerramientaFinal\WObj:=Workobject_Final;
        MoveC Target_220,Target_230, v100,z1,HerramientaFinal\WObj:=Workobject_Final;
        MoveL Target_240,v100,z1,HerramientaFinal\WObj:=Workobject_Final;
        MoveL Target_250,v100,z1,HerramientaFinal\WObj:=Workobject_Final;
        MoveC Target_260,Target_270,v100,z1,HerramientaFinal\WObj:=Workobject_Final;
        MoveL Target_280,v100,z1,HerramientaFinal\WObj:=Workobject_Final;
        MoveL Target_290,v100,z1,HerramientaFinal\WObj:=Workobject_Final;
        MoveL Target_190,v100,z1,HerramientaFinal\WObj:=Workobject_Final;
    ENDPROC
    PROC Path_U()
        MoveJ Target_300,v200,z1,HerramientaFinal\WObj:=Workobject_Final;
        MoveL Target_310,v100,z1,HerramientaFinal\WObj:=Workobject_Final;
        MoveL Target_320,v100,z1,HerramientaFinal\WObj:=Workobject_Final;
        MoveL Target_330,v100,z1,HerramientaFinal\WObj:=Workobject_Final;
        MoveC Target_340,Target_350,v100,z1,HerramientaFinal\WObj:=Workobject_Final;
        MoveC Target_360,Target_370,v100,z1,HerramientaFinal\WObj:=Workobject_Final;
        MoveL Target_380,v100,z1,HerramientaFinal\WObj:=Workobject_Final;
        MoveL Target_390,v100,z1,HerramientaFinal\WObj:=Workobject_Final;
        MoveL Target_400,v100,z10,HerramientaFinal\WObj:=Workobject_Final;
        MoveC Target_410,Target_420,v100,z1,HerramientaFinal\WObj:=Workobject_Final;
        MoveC Target_430,Target_440,v100,z1,HerramientaFinal\WObj:=Workobject_Final;
        MoveL Target_310,v100,z1,HerramientaFinal\WObj:=Workobject_Final;





    ENDPROC
    PROC Path_A()
        MoveJ Target_450,v200,z1,HerramientaFinal\WObj:=Workobject_Final;
        MoveL Target_460,v100,z1,HerramientaFinal\WObj:=Workobject_Final;
        MoveL Target_470,v100,z1,HerramientaFinal\WObj:=Workobject_Final;
        MoveL Target_480,v100,z1,HerramientaFinal\WObj:=Workobject_Final;
        MoveL Target_490,v100,z1,HerramientaFinal\WObj:=Workobject_Final;
        MoveL Target_500,v100,z1,HerramientaFinal\WObj:=Workobject_Final;
        MoveL Target_510,v100,z1,HerramientaFinal\WObj:=Workobject_Final;
        MoveL Target_520,v100,z1,HerramientaFinal\WObj:=Workobject_Final;
        MoveL Target_530,v100,z1,HerramientaFinal\WObj:=Workobject_Final;
        MoveL Target_460,v100,z1,HerramientaFinal\WObj:=Workobject_Final;
        MoveJ Target_540,v100,z1,HerramientaFinal\WObj:=Workobject_Final;
        MoveL Target_550,v100,z1,HerramientaFinal\WObj:=Workobject_Final;
        MoveL Target_560,v100,z1,HerramientaFinal\WObj:=Workobject_Final;
        MoveL Target_570,v100,z1,HerramientaFinal\WObj:=Workobject_Final;
        MoveL Target_550,v100,z1,HerramientaFinal\WObj:=Workobject_Final;
    ENDPROC
    PROC Path_N()
        MoveJ Target_580,v200,z1,HerramientaFinal\WObj:=Workobject_Final;
        MoveL Target_590,v100,z1,HerramientaFinal\WObj:=Workobject_Final;
        MoveL Target_600,v100,z1,HerramientaFinal\WObj:=Workobject_Final;
        MoveL Target_610,v100,z1,HerramientaFinal\WObj:=Workobject_Final;
        MoveL Target_620,v100,z1,HerramientaFinal\WObj:=Workobject_Final;
        MoveL Target_630,v100,z1,HerramientaFinal\WObj:=Workobject_Final;
        MoveL Target_640,v100,z1,HerramientaFinal\WObj:=Workobject_Final;
        MoveL Target_650,v100,z1,HerramientaFinal\WObj:=Workobject_Final;
        MoveL Target_660,v100,z1,HerramientaFinal\WObj:=Workobject_Final;
        MoveL Target_670,v100,z1,HerramientaFinal\WObj:=Workobject_Final;
        MoveL Target_680,v100,z1,HerramientaFinal\WObj:=Workobject_Final;
        MoveL Target_590,v100,z1,HerramientaFinal\WObj:=Workobject_Final;
    ENDPROC
    PROC Path_M()
        MoveJ Target_690,v200,z1,HerramientaFinal\WObj:=Workobject_Final;
        MoveL Target_700,v100,z1,HerramientaFinal\WObj:=Workobject_Final;
        MoveL Target_710,v100,z1,HerramientaFinal\WObj:=Workobject_Final;
        MoveL Target_720,v100,z1,HerramientaFinal\WObj:=Workobject_Final;
        MoveL Target_730,v100,z1,HerramientaFinal\WObj:=Workobject_Final;
        MoveL Target_740,v100,z1,HerramientaFinal\WObj:=Workobject_Final;
        MoveL Target_750,v100,z1,HerramientaFinal\WObj:=Workobject_Final;
        MoveL Target_760,v100,z1,HerramientaFinal\WObj:=Workobject_Final;
        MoveL Target_770,v100,z1,HerramientaFinal\WObj:=Workobject_Final;
        MoveL Target_780,v100,z1,HerramientaFinal\WObj:=Workobject_Final;
        MoveL Target_790,v100,z1,HerramientaFinal\WObj:=Workobject_Final;
        MoveL Target_800,v100,z1,HerramientaFinal\WObj:=Workobject_Final;
        MoveL Target_810,v100,z1,HerramientaFinal\WObj:=Workobject_Final;
        MoveL Target_820,v100,z1,HerramientaFinal\WObj:=Workobject_Final;
        MoveL Target_700,v100,z1,HerramientaFinal\WObj:=Workobject_Final;
    ENDPROC
    PROC Path_A2()
        MoveL Target_830,v200,z1,HerramientaFinal\WObj:=Workobject_Final;
        MoveL Target_840,v100,z1,HerramientaFinal\WObj:=Workobject_Final;
        MoveL Target_850,v100,z1,HerramientaFinal\WObj:=Workobject_Final;
        MoveL Target_860,v100,z1,HerramientaFinal\WObj:=Workobject_Final;
        MoveL Target_870,v100,z1,HerramientaFinal\WObj:=Workobject_Final;
        MoveL Target_880,v100,z1,HerramientaFinal\WObj:=Workobject_Final;
        MoveL Target_890,v100,z1,HerramientaFinal\WObj:=Workobject_Final;
        MoveL Target_900,v100,z1,HerramientaFinal\WObj:=Workobject_Final;
        MoveL Target_910,v100,z1,HerramientaFinal\WObj:=Workobject_Final;
        MoveL Target_840,v100,z1,HerramientaFinal\WObj:=Workobject_Final;
        MoveJ Target_920,v100,z1,HerramientaFinal\WObj:=Workobject_Final;
        MoveL Target_930,v100,z1,HerramientaFinal\WObj:=Workobject_Final;
        MoveL Target_940,v100,z1,HerramientaFinal\WObj:=Workobject_Final;
        MoveL Target_950,v100,z1,HerramientaFinal\WObj:=Workobject_Final;
        MoveL Target_930,v100,z1,HerramientaFinal\WObj:=Workobject_Final;
    ENDPROC
    PROC Path_T()
        MoveJ Target_960,v200,z1,HerramientaFinal\WObj:=Workobject_Final;
        MoveL Target_970,v100,z1,HerramientaFinal\WObj:=Workobject_Final;
        MoveL Target_980,v100,z1,HerramientaFinal\WObj:=Workobject_Final;
        MoveL Target_990,v100,z1,HerramientaFinal\WObj:=Workobject_Final;
        MoveL Target_1000,v100,z1,HerramientaFinal\WObj:=Workobject_Final;
        MoveL Target_1010,v100,z1,HerramientaFinal\WObj:=Workobject_Final;
        MoveL Target_1020,v100,z1,HerramientaFinal\WObj:=Workobject_Final;
        MoveL Target_1030,v100,z1,HerramientaFinal\WObj:=Workobject_Final;
        MoveL Target_1040,v100,z1,HerramientaFinal\WObj:=Workobject_Final;
        MoveL Target_970,v100,z1,HerramientaFinal\WObj:=Workobject_Final;
    ENDPROC
    PROC Path_E()
        MoveJ Target_1050,v200,z1,HerramientaFinal\WObj:=Workobject_Final;
        MoveL Target_1060,v100,z1,HerramientaFinal\WObj:=Workobject_Final;
        MoveL Target_1070,v100,z1,HerramientaFinal\WObj:=Workobject_Final;
        MoveL Target_1080,v100,z1,HerramientaFinal\WObj:=Workobject_Final;
        MoveL Target_1090,v100,z1,HerramientaFinal\WObj:=Workobject_Final;
        MoveL Target_1100,v100,z1,HerramientaFinal\WObj:=Workobject_Final;
        MoveL Target_1110,v100,z1,HerramientaFinal\WObj:=Workobject_Final;
        MoveL Target_1120,v100,z1,HerramientaFinal\WObj:=Workobject_Final;
        MoveL Target_1130,v100,z1,HerramientaFinal\WObj:=Workobject_Final;
        MoveL Target_1140,v100,z1,HerramientaFinal\WObj:=Workobject_Final;
        MoveL Target_1150,v100,z1,HerramientaFinal\WObj:=Workobject_Final;
        MoveL Target_1160,v100,z1,HerramientaFinal\WObj:=Workobject_Final;
        MoveL Target_1170,v100,z1,HerramientaFinal\WObj:=Workobject_Final;
        MoveL Target_1060,v100,z1,HerramientaFinal\WObj:=Workobject_Final;
    ENDPROC
    PROC Path_0()
        MoveJ Target_1180,v200,z1,HerramientaFinal\WObj:=Workobject_Final;
        MoveL Target_1190,v100,z1,HerramientaFinal\WObj:=Workobject_Final;
        MoveC Target_1200,Target_1210,v100,z1,HerramientaFinal\WObj:=Workobject_Final;
        MoveL Target_1220,v100,z1,HerramientaFinal\WObj:=Workobject_Final;
        MoveC Target_1230,Target_1240,v100,z1,HerramientaFinal\WObj:=Workobject_Final;
        MoveC Target_1250,Target_1260,v100,z1,HerramientaFinal\WObj:=Workobject_Final;
        MoveL Target_1270,v100,z1,HerramientaFinal\WObj:=Workobject_Final;
        MoveC Target_1280,Target_1190,v100,z1,HerramientaFinal\WObj:=Workobject_Final;
        MoveJ Target_1290,v100,z1,HerramientaFinal\WObj:=Workobject_Final;
        MoveL Target_1300,v100,z1,HerramientaFinal\WObj:=Workobject_Final;
        MoveC Target_1310,Target_1320,v100,z1,HerramientaFinal\WObj:=Workobject_Final;
        MoveL Target_1330,v100,z1,HerramientaFinal\WObj:=Workobject_Final;
        MoveC Target_1340,Target_1350,v100,z1,HerramientaFinal\WObj:=Workobject_Final;
        MoveC Target_1360,Target_1370,v100,z1,HerramientaFinal\WObj:=Workobject_Final;
        MoveL Target_1380,v100,z1,HerramientaFinal\WObj:=Workobject_Final;
        MoveC Target_1390,Target_1300,v100,z1,HerramientaFinal\WObj:=Workobject_Final;

    ENDPROC
    PROC Path_SansBorde()
        MoveJ Target_1400,v200,z1,HerramientaFinal\WObj:=Workobject_Final;
        MoveL Target_1410,v100,z1,HerramientaFinal\WObj:=Workobject_Final;

        MoveC Target_1420,Target_1430,v100,z1,HerramientaFinal\WObj:=Workobject_Final;
        MoveC Target_1440,Target_1450,v100,z1,HerramientaFinal\WObj:=Workobject_Final;
        MoveC Target_1460,Target_1470,v100,z1,HerramientaFinal\WObj:=Workobject_Final;
        MoveC Target_1480,Target_1490,v100,z1,HerramientaFinal\WObj:=Workobject_Final;
        MoveC Target_1500,Target_1510,v100,z1,HerramientaFinal\WObj:=Workobject_Final;
        MoveC Target_1520,Target_1410,v100,z1,HerramientaFinal\WObj:=Workobject_Final;

    ENDPROC
    PROC Path_Sans_OJO1()
        MoveJ Target_1530,v200,z1,HerramientaFinal\WObj:=Workobject_Final;
        MoveL Target_1540,v100,z1,HerramientaFinal\WObj:=Workobject_Final;
        MoveC Target_1550,Target_1560,v100,z1,HerramientaFinal\WObj:=Workobject_Final;
        MoveC Target_1570,Target_1580,v100,z1,HerramientaFinal\WObj:=Workobject_Final;
        MoveC Target_1590,Target_1600,v100,z1,HerramientaFinal\WObj:=Workobject_Final;
        MoveC Target_1610,Target_1540,v100,z1,HerramientaFinal\WObj:=Workobject_Final;
    ENDPROC
    PROC Path_Sans_OJO2()
        MoveJ Target_1620,v200,z1,HerramientaFinal\WObj:=Workobject_Final;
        MoveL Target_1630,v100,z1,HerramientaFinal\WObj:=Workobject_Final;
        MoveC Target_1640,Target_1650,v100,z1,HerramientaFinal\WObj:=Workobject_Final;
        MoveC Target_1660,Target_1670,v100,z1,HerramientaFinal\WObj:=Workobject_Final;
        MoveC Target_1680,Target_1630,v100,z1,HerramientaFinal\WObj:=Workobject_Final;
    ENDPROC
    PROC Path_SansBoca()
        MoveJ Target_1690,v200,z1,HerramientaFinal\WObj:=Workobject_Final;
        MoveL Target_1700,v100,z1,HerramientaFinal\WObj:=Workobject_Final;
        MoveC Target_1710,Target_1720,v100,z1,HerramientaFinal\WObj:=Workobject_Final;
        MoveC Target_1730,Target_1740,v100,z1,HerramientaFinal\WObj:=Workobject_Final;
        MoveC Target_1750,Target_1760,v100,z1,HerramientaFinal\WObj:=Workobject_Final;
        MoveC Target_1770,Target_1780,v100,z1,HerramientaFinal\WObj:=Workobject_Final;
        MoveC Target_1790,Target_1700,v100,z1,HerramientaFinal\WObj:=Workobject_Final;
    ENDPROC
    PROC Path_SansPUPILA1()
        MoveJ Target_1800,v200,z1,HerramientaFinal\WObj:=Workobject_Final;
        MoveL Target_1810,v100,z1,HerramientaFinal\WObj:=Workobject_Final;
        MoveC Target_1820,Target_1830,v100,z1,HerramientaFinal\WObj:=Workobject_Final;
        MoveC Target_1840,Target_1810,v100,z1,HerramientaFinal\WObj:=Workobject_Final;
    ENDPROC
    PROC Path_SansPUPILA2()
        MoveJ Target_1850,v200,z1,HerramientaFinal\WObj:=Workobject_Final;
        MoveL Target_1860,v100,z1,HerramientaFinal\WObj:=Workobject_Final;
        MoveC Target_1870,Target_1880,v100,z1,HerramientaFinal\WObj:=Workobject_Final;
        MoveC Target_1890,Target_1860,v100,z1,HerramientaFinal\WObj:=Workobject_Final;
    ENDPROC
    PROC Path_SansNariz()
        MoveJ Target_1900,v200,z1,HerramientaFinal\WObj:=Workobject_Final;
        MoveL Target_1910,v100,z1,HerramientaFinal\WObj:=Workobject_Final;
        MoveC Target_1920,Target_1930,v100,z1,HerramientaFinal\WObj:=Workobject_Final;
        MoveC Target_1940,Target_1950,v100,z1,HerramientaFinal\WObj:=Workobject_Final;
        MoveC Target_1960,Target_1970,v100,z1,HerramientaFinal\WObj:=Workobject_Final;
        MoveC Target_1980,Target_1990,v100,z1,HerramientaFinal\WObj:=Workobject_Final;
        MoveC Target_2000,Target_2010,v100,z1,HerramientaFinal\WObj:=Workobject_Final;
        MoveC Target_2020,Target_1910,v100,z1,HerramientaFinal\WObj:=Workobject_Final;
    ENDPROC
    PROC Path_SansDientes()
        MoveJ Target_2030,v200,z1,HerramientaFinal\WObj:=Workobject_Final;
        MoveL Target_2040,v100,z1,HerramientaFinal\WObj:=Workobject_Final;
        MoveL Target_2050,v100,z1,HerramientaFinal\WObj:=Workobject_Final;
        MoveJ Target_2060,v200,z1,HerramientaFinal\WObj:=Workobject_Final;
        MoveL Target_2070,v100,z1,HerramientaFinal\WObj:=Workobject_Final;
        MoveL Target_2070B,v100,z1,HerramientaFinal\WObj:=Workobject_Final;
        MoveJ Target_2080,v200,z1,HerramientaFinal\WObj:=Workobject_Final;
        MoveL Target_2090,v100,z1,HerramientaFinal\WObj:=Workobject_Final;
        MoveL Target_2100,v100,z1,HerramientaFinal\WObj:=Workobject_Final;
        MoveJ Target_2110,v200,z1,HerramientaFinal\WObj:=Workobject_Final;
        MoveL Target_2120,v100,z1,HerramientaFinal\WObj:=Workobject_Final;
        MoveL Target_2130,v100,z1,HerramientaFinal\WObj:=Workobject_Final;
        MoveJ Target_2140,v200,z1,HerramientaFinal\WObj:=Workobject_Final;
        MoveL Target_2150,v100,z1,HerramientaFinal\WObj:=Workobject_Final;
        MoveL Target_2160,v100,z1,HerramientaFinal\WObj:=Workobject_Final;
    ENDPROC
    PROC Path_Mantenimiento()
        MoveJ Target_Mantenimiento,v100,z100,HerramientaFinal\WObj:=Workobject_Final;
    ENDPROC
    PROC Path_Mantenimiento2()
        MoveL Target_10,v200,z100,HerramientaFinal\WObj:=Workobject_Final;
        MoveJ Target_Mantenimiento,v100,z100,HerramientaFinal\WObj:=Workobject_Final;
    ENDPROC
ENDMODULE
